// LS Electric XG5000 project: 신호등
// PLC LSPLC

PROGRAM NewProgram (task: 스캔 프로그램)

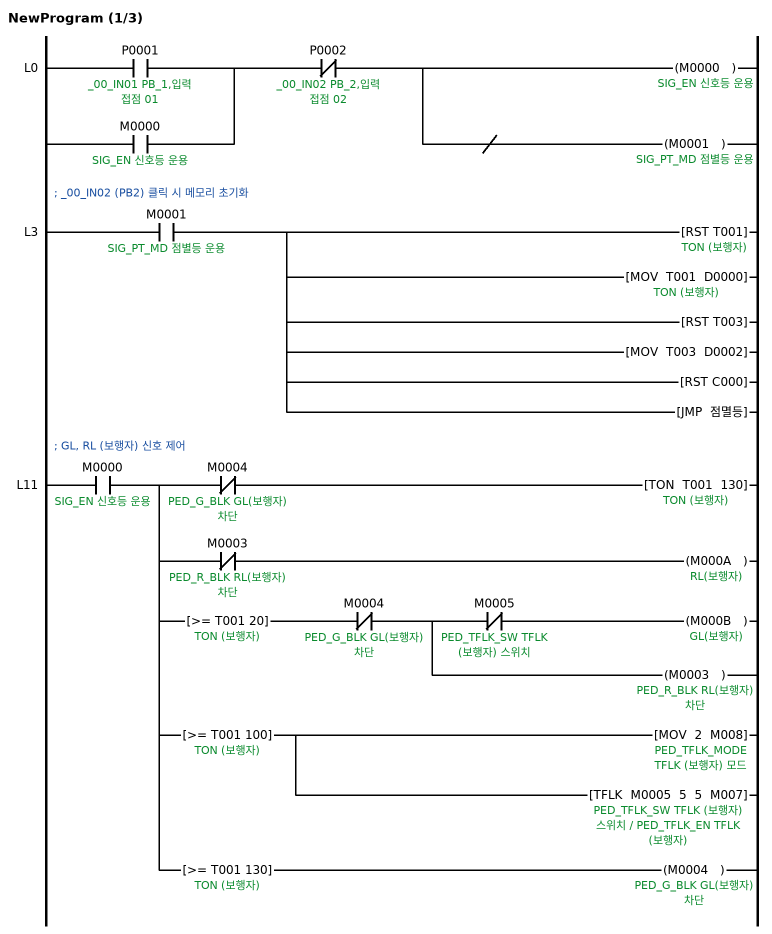
; L0
LOAD      P0001	// _00_IN01 PB_1,입력 접점 01
OR        M0000	// SIG_EN 신호등 운용
AND NOT   P0002	// _00_IN02 PB_2,입력 접점 02
OUT       M0000	// SIG_EN 신호등 운용
NOT
OUT       M0001	// SIG_PT_MD 점별등 운용
//  _00_IN02 (PB2) 클릭 시 메모리 초기화
; L3
LOAD      M0001	// SIG_PT_MD 점별등 운용
RST       T001	// TON (보행자)
MOV       T001 D0000	// TON (보행자)
RST       T003
MOV       T003 D0002
RST       C000
JMP       점멸등
//  GL, RL (보행자) 신호 제어
; L11
LOAD      M0000	// SIG_EN 신호등 운용
MPUSH
AND NOT   M0004	// PED_G_BLK GL(보행자) 차단
TON       T001 130	// TON (보행자)
MLOAD
AND NOT   M0003	// PED_R_BLK RL(보행자) 차단
OUT       M000A	// RL(보행자)
MLOAD
AND>=     T001 20	// TON (보행자)
AND NOT   M0004	// PED_G_BLK GL(보행자) 차단
MPUSH
AND NOT   M0005	// PED_TFLK_SW TFLK (보행자) 스위치
OUT       M000B	// GL(보행자)
MPOP
OUT       M0003	// PED_R_BLK RL(보행자) 차단
MLOAD
AND>=     T001 100	// TON (보행자)
MOV       2 M008	// PED_TFLK_MODE TFLK (보행자) 모드
TFLK      M0005 5 5 M007	// PED_TFLK_SW TFLK (보행자) 스위치 / PED_TFLK_EN TFLK (보행자)
MPOP
AND>=     T001 130	// TON (보행자)
OUT       M0004	// PED_G_BLK GL(보행자) 차단

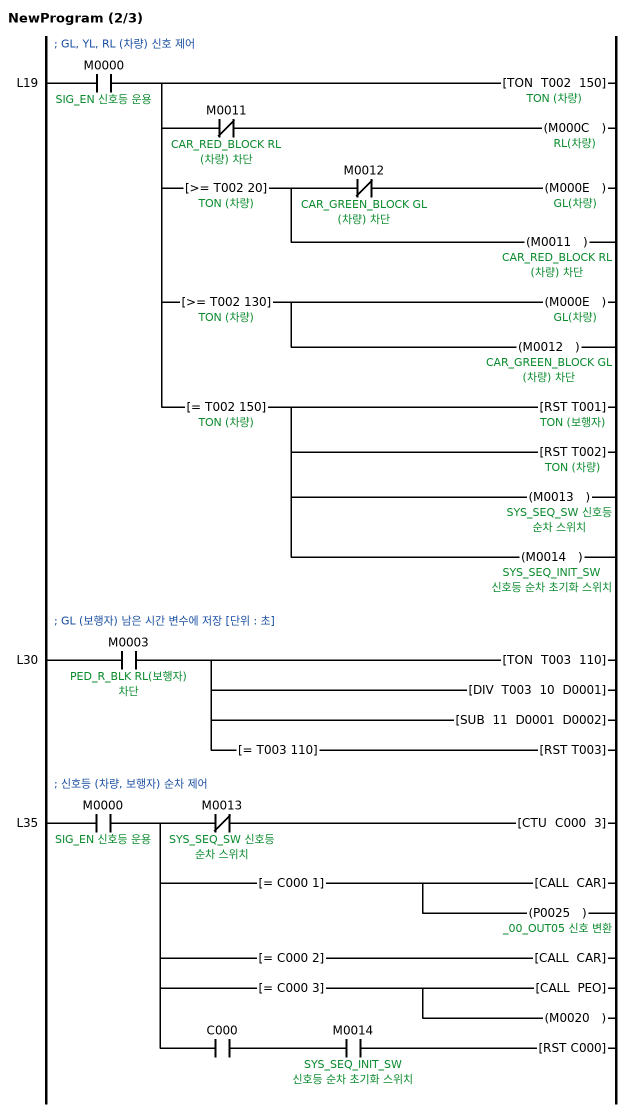
//  GL, YL, RL (차량) 신호 제어
; L19
LOAD      M0000	// SIG_EN 신호등 운용
TON       T002 150	// TON (차량)
MPUSH
AND NOT   M0011	// CAR_RED_BLOCK RL (차량) 차단
OUT       M000C	// RL(차량)
MLOAD
AND>=     T002 20	// TON (차량)
MPUSH
AND NOT   M0012	// CAR_GREEN_BLOCK GL (차량) 차단
OUT       M000E	// GL(차량)
MPOP
OUT       M0011	// CAR_RED_BLOCK RL (차량) 차단
MLOAD
AND>=     T002 130	// TON (차량)
OUT       M000E	// GL(차량)
OUT       M0012	// CAR_GREEN_BLOCK GL (차량) 차단
MPOP
AND=      T002 150	// TON (차량)
RST       T001	// TON (보행자)
RST       T002	// TON (차량)
OUT       M0013	// SYS_SEQ_SW 신호등 순차 스위치
OUT       M0014	// SYS_SEQ_INIT_SW 신호등 순차 초기화 스위치
//  GL (보행자) 남은 시간 변수에 저장 [단위 : 초]
; L30
LOAD      M0003	// PED_R_BLK RL(보행자) 차단
TON       T003 110
DIV       T003 10 D0001
SUB       11 D0001 D0002
AND=      T003 110
RST       T003
//  신호등 (차량, 보행자) 순차 제어
; L35
LOAD      M0000	// SIG_EN 신호등 운용
MPUSH
AND NOT   M0013	// SYS_SEQ_SW 신호등 순차 스위치
CTU       C000 3
MLOAD
AND=      C000 1
CALL      CAR
OUT       P0025	// _00_OUT05 신호 변환
MLOAD
AND=      C000 2
CALL      CAR
MLOAD
AND=      C000 3
CALL      PEO
OUT       M0020
MPOP
AND       C000
AND       M0014	// SYS_SEQ_INIT_SW 신호등 순차 초기화 스위치
RST       C000

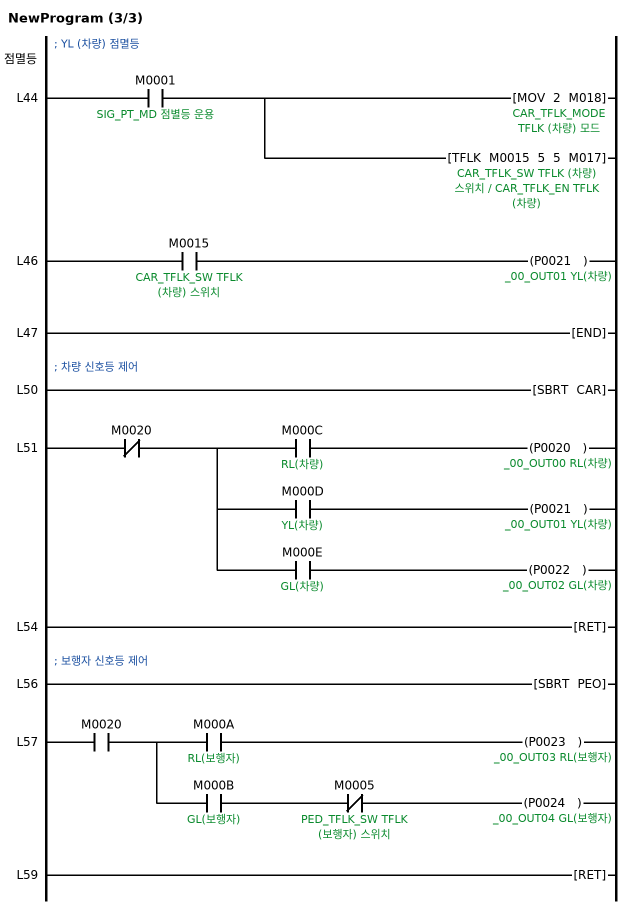
//  YL (차량) 점멸등
점멸등:
; L44
LOAD      M0001	// SIG_PT_MD 점별등 운용
MOV       2 M018	// CAR_TFLK_MODE TFLK (차량) 모드
TFLK      M0015 5 5 M017	// CAR_TFLK_SW TFLK (차량) 스위치 / CAR_TFLK_EN TFLK (차량)
; L46
LOAD      M0015	// CAR_TFLK_SW TFLK (차량) 스위치
OUT       P0021	// _00_OUT01 YL(차량)
; L47
END
// 차량 신호등 제어
; L50
SBRT      CAR
; L51
LOAD NOT  M0020
MPUSH
AND       M000C	// RL(차량)
OUT       P0020	// _00_OUT00 RL(차량)
MLOAD
AND       M000D	// YL(차량)
OUT       P0021	// _00_OUT01 YL(차량)
MPOP
AND       M000E	// GL(차량)
OUT       P0022	// _00_OUT02 GL(차량)
; L54
RET
// 보행자 신호등 제어
; L56
SBRT      PEO
; L57
LOAD      M0020
MPUSH
AND       M000A	// RL(보행자)
OUT       P0023	// _00_OUT03 RL(보행자)
MPOP
AND       M000B	// GL(보행자)
AND NOT   M0005	// PED_TFLK_SW TFLK (보행자) 스위치
OUT       P0024	// _00_OUT04 GL(보행자)
; L59
RET